PROGRAM MAIN
VAR
END_VAR

//ergänzung 1
//ergänzung 2

END_PROGRAM

(* stored: Version 1.1.0.1, ProductVersion 3.1.4020.12
   POU MAIN: Id {237c6c83-1484-4b26-bbd7-d367abb321c0}, SpecialFunc None *)
